FUNCTION_BLOCK E_RESTART
  (* Version 0.1, 2005-04-08, Goran, Chalmers *)
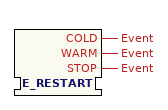
  EVENT_OUTPUT
    COLD;
    WARM;
    STOP;
  END_EVENT
END_FUNCTION_BLOCK
